FUNCTION_BLOCK FB_MatAndToolHandling EXTENDS FB_CompositionBase
VAR
	
	// Sequencer
	fbSeq						: FB_Sequence;
	
	stPosition					: ST_Coordinate;
	nToolDockingNr				: INT;
	
	fVelocityX					: LREAL;	
	fVelocityY					: LREAL;
	fAccelerationX				: LREAL;	
	fAccelerationY				: LREAL;
	
	bJogReverseDirectionX		: BOOL;
	bJogReverseDirectionY		: BOOL;
	bJogX						: BOOL;
	bJogY						: BOOL;
		
	bMoveX						: BOOL;
	bMoveY						: BOOL;
	
	// Watch Variables	
	refObstacle					: REFERENCE TO BOOL;
	bInPosition					: BOOL;
	
	// Tool/Mat Data
	nCurTooldockingNr			: INT;
	afDistanceTooldocking		: ARRAY[1..2] OF REAL;	
	astOffsetDie				: ARRAY[1..2] OF ST_Coordinate;
	

	nVelocityMultiplier			: INT;
	nAccelerationMultiplier		: INT;	
	stOffsetMat					: ST_Coordinate;
	
	
	// Settings
	
	fMaxVelocityX				: LREAL;
	fMinVelocityX				: LREAL;
	fMaxAccelerationX			: LREAL;
	fMinAccelerationX			: LREAL;
	
	fMaxVelocityY				: LREAL;
	fMinVelocityY				: LREAL;
	fMaxAccelerationY			: LREAL;
	fMinAccelerationY			: LREAL;
	
	fDefaultVelocity			: LREAL;
	fDefaultAcceleration		: LREAL;	
	
	fToleranceWindow			: LREAL := 0.5;
	stMaintPosition				: ST_Coordinate;
	
	// Axis
	bEnable						: BOOL := TRUE;
	refEnable					: REFERENCE TO BOOL;
	fbAxisX						: FB_AxisDriver;
	fbAxisY						: FB_AxisDriver;
	
	// Cylinder
	fbToolSelector				: FB_CylinderDriver;
	
END_VAR

METHOD _ChangeTool : BOOL
VAR_INPUT
END_VAR
fbSeq.Name := 'ChangeTool';

CASE fbSeq.Step OF
	

0	 :	fbSeq.StepDefinition('switch Valves for selected Tooldocking', T#0S);
		
		CASE nToolDockingNr OF
			1: fbToolSelector.ToWP();		
			2: fbToolSelector.ToHP();
		END_CASE

		fbSeq.NextStep(10);
	
	
10	 :	fbSeq.StepDefinition('Tooldock changing', T#0S);

		IF fbToolSelector.ActualPosition = fbToolSelector.RequestPosition THEN
			nCurTooldockingNr := nToolDockingNr;
			fbSeq.Finish();
		END_IF
	

END_CASE
END_METHOD

METHOD _Halt : BOOL
VAR_INPUT
END_VAR
fbSeq.Name := 'Halt';

CASE fbSeq.Step OF
	

0	 :	fbSeq.StepDefinition('Punchaxis Halt', T#0S);
		fbAxisX.Halt();
		fbAxisY.Halt();				
		fbSeq.NextStep(10);
	
	
10	 :	fbSeq.StepDefinition('', T#0S);
		IF fbAxisX.NotMoving AND fbAxisY.NotMoving THEN
			fbSeq.Finish();
		END_IF
	
END_CASE
END_METHOD

METHOD _Homeing : BOOL
VAR_INPUT
END_VAR
fbSeq.Name := 'Homeing';

CASE fbSeq.Step OF
	

0	 :	fbSeq.StepDefinition('', T#0S);

		fbSeq.NextStep(10);
	
	
10	 :	fbSeq.StepDefinition('', T#0S);

		fbSeq.NextStep(20);	

		
20	 :	fbSeq.StepDefinition('', T#0S);

		fbSeq.NextStep(30);	

		
30	 :	fbSeq.StepDefinition('', T#0S);

		fbSeq.NextStep(40);

		
40	 :	fbSeq.StepDefinition('', T#0S);

		fbSeq.NextStep(50);

		
50	 :	fbSeq.StepDefinition('', T#0S);

		fbSeq.Finish();

END_CASE
END_METHOD

METHOD _Jog : BOOL
VAR
	
END_VAR
fbSeq.Name := 'Jog';

CASE fbSeq.Step OF
	

0	 :	fbSeq.StepDefinition('Halt Axis', T#0S);
		fbAxisX.Halt();
		fbAxisY.Halt();	
		fbSeq.NextStep(10);
	
10	 :	fbSeq.StepDefinition('Jog Axis', T#0S);
	
		IF bJogX OR bJogY THEN
			fbAxisX.JogAcc(bJogX AND NOT bJogReverseDirectionX , bJogX AND bJogReverseDirectionX);
			fbAxisY.JogAcc(bJogY AND NOT bJogReverseDirectionY , bJogY AND bJogReverseDirectionY);
		ELSE
			fbSeq.NextStep(20);
		END_IF		
		
20	 :	fbSeq.StepDefinition('Jog Finish', T#0S);
		fbAxisX.Halt();
		fbAxisY.Halt();	
		fbSeq.Finish();

END_CASE
END_METHOD

METHOD _MoveAbs : BOOL
VAR
	stMovAbsParameter			: ST_AxisMoveAbsParameter;
END_VAR
fbSeq.Name := 'MoveAbs';

CASE fbSeq.Step OF
	

0	 :	fbSeq.StepDefinition('Move Axis to Position', T#0S);
		
		IF bMoveX THEN
			stMovAbsParameter.fAcceleration := fAccelerationX;
			stMovAbsParameter.fDeceleration := fAccelerationX;
			stMovAbsParameter.fVelocity := fVelocityX;
			stMovAbsParameter.fPosition := stPosition.fX;
			fbAxisX.MoveAbsEx(stMovAbsParameter);
		END_IF
			
		IF bMoveY THEN
			stMovAbsParameter.fAcceleration := fAccelerationY;
			stMovAbsParameter.fDeceleration := fAccelerationY;
			stMovAbsParameter.fVelocity := fVelocityY;
			stMovAbsParameter.fPosition := stPosition.fY;
			fbAxisY.MoveAbsEx(stMovAbsParameter);
		END_IF
		
		fbSeq.NextStep(20);	
		
20	 :	fbSeq.StepDefinition('Axis moving', T#0S);
		IF (fbAxisX.TargetReached(fToleranceWindow) OR NOT bMoveX) AND (fbAxisY.TargetReached(fToleranceWindow) OR NOT bMoveY) THEN
			fbSeq.Finish();
		END_IF

END_CASE
END_METHOD

/// Actual amplifier temp. [°C]
PROPERTY AmplifierTemp : LREAL
GET
/// Actual amplifier temp. [°C]
AmplifierTemp := MAX(fbAxisX.AmplifierTemp, fbAxisY.AmplifierTemp);
END_GET
END_PROPERTY

METHOD ChangeTool : E_OperationResult
VAR_INPUT
	ToolDockingNr				: INT;
END_VAR
// init result pessimistic
ChangeTool := E_OperationResult.eOperationResult_NOk;

bInPosition := FALSE;


stPosition := stMaintPosition;
fVelocityX := fVelocityY := fDefaultVelocity;	
fAccelerationX := fAccelerationY := fDefaultAcceleration;
nToolDockingNr := ToolDockingNr;
bMoveX := TRUE;
bMoveY := TRUE;

fbSeq.Start(E_MatAndToolHandlingCmd.cmdChangeTool);

ChangeTool := E_OperationResult.eOperationResult_Ok;
END_METHOD

PROPERTY CurTool : INT
GET
CurTool := nCurTooldockingNr;
END_GET
END_PROPERTY

METHOD FB_init : BOOL
VAR_INPUT
	bInitRetains : BOOL; // if TRUE, the retain variables are initialized (warm start / cold start)
	bInCopyCode : BOOL;  // if TRUE, the instance afterwards gets moved into the copy code (online change)
END_VAR
eTyp := E_ComponentType.eComponentType_MatAndToolHandling;
END_METHOD

METHOD GetMovementTime : LREAL
VAR_INPUT
	DistanceX		: LREAL;
	DistanceY		: LREAL;
	VelocityX		: LREAL;
	AccelerationX	: LREAL;
	VelocityY		: LREAL;
	AccelerationY	: LREAL;
END_VAR
VAR
	tmpTimeX		: LREAL;
	tmpTimeY		: LREAL;
	
	tmpTimeB		: LREAL;
	tmpTimeBB		: LREAL;
END_VAR
// X
tmpTimeB  := VelocityX/AccelerationX;
tmpTimeBB := 2*SQRT(DistanceX/AccelerationX);

IF tmpTimeBB/2 > tmpTimeB THEN
	tmpTimeX := DistanceX/VelocityX + VelocityX/AccelerationX;
ELSE
	tmpTimeX := tmpTimeBB;
END_IF


// Y
tmpTimeB  := VelocityY/AccelerationY;
tmpTimeBB := 2*SQRT(DistanceY/AccelerationY);

IF tmpTimeBB/2 > tmpTimeB THEN
	tmpTimeY := DistanceY/fVelocityY + VelocityY/AccelerationY;
ELSE
	tmpTimeY := tmpTimeBB;
END_IF


GetMovementTime := MAX(tmpTimeX, tmpTimeY)*1.2;	// 20% sicherheit
END_METHOD

METHOD Halt : E_OperationResult
VAR_INPUT
END_VAR
// init result pessimistic
Halt := E_OperationResult.eOperationResult_NOk;

bInPosition := FALSE;


fVelocityX := fVelocityY := fDefaultVelocity;	
fAccelerationX := fAccelerationY := fDefaultAcceleration;
bMoveX := FALSE;
bMoveY := FALSE;

fbSeq.Start(E_MatAndToolHandlingCmd.cmdHalt);

Halt := E_OperationResult.eOperationResult_Ok;
END_METHOD

PROPERTY Homed : BOOL
GET
Homed := fbaxisX.Homed AND fbaxisY.Homed;
END_GET
END_PROPERTY

METHOD Homing : E_OperationResult
VAR_INPUT
END_VAR
// init result pessimistic
Homing := E_OperationResult.eOperationResult_NOk;

bInPosition := FALSE;


stPosition := stMaintPosition;
fVelocityX := fVelocityY := fDefaultVelocity;	
fAccelerationX := fAccelerationY := fDefaultAcceleration;
bMoveX := TRUE;
bMoveY := TRUE;

fbSeq.Start(E_MatAndToolHandlingCmd.cmdHomeing);

Homing := E_OperationResult.eOperationResult_Ok;
END_METHOD

METHOD JogX : E_OperationResult
VAR_INPUT
	ReverseDirection					: BOOL;
END_VAR
// init result pessimistic
JogX := E_OperationResult.eOperationResult_NOk;
bInPosition := FALSE;

IF fbSeq.SequenceId <> E_MatAndToolHandlingCmd.cmdJog THEN
	fbSeq.Start(E_MatAndToolHandlingCmd.cmdJog);
//	RETURN;
END_IF


bJogReverseDirectionX := ReverseDirection;
bJogX := TRUE;	

JogX := E_OperationResult.eOperationResult_Ok;
END_METHOD

METHOD JogXStop : E_OperationResult
VAR_INPUT
END_VAR
// init result pessimistic
JogXStop := E_OperationResult.eOperationResult_NOk;

bJogX := FALSE;	

JogXStop := E_OperationResult.eOperationResult_Ok;
END_METHOD

METHOD JogY : E_OperationResult
VAR_INPUT
	ReverseDirection					: BOOL;
END_VAR
// init result pessimistic
JogY := E_OperationResult.eOperationResult_NOk;
bInPosition := FALSE;

IF fbSeq.SequenceId <> E_MatAndToolHandlingCmd.cmdJog THEN
	fbSeq.Start(E_MatAndToolHandlingCmd.cmdJog);
//	RETURN;
END_IF


bJogReverseDirectionY := ReverseDirection;
bJogY := TRUE;	

JogY := E_OperationResult.eOperationResult_Ok;
END_METHOD

METHOD JogYStop : E_OperationResult
VAR_INPUT
END_VAR
// init result pessimistic
JogYStop := E_OperationResult.eOperationResult_NOk;

bJogY := FALSE;	

JogYStop := E_OperationResult.eOperationResult_Ok;
END_METHOD

METHOD MaintPos : E_OperationResult
VAR_INPUT
	bXOnly				: BOOL;
	bYOnly				: BOOL;
END_VAR
IF bXOnly THEN
	MaintPos := MoveAbsX(stMaintPosition.fX,fDefaultVelocity, fDefaultAcceleration);	
ELSIF bYOnly THEN
	MaintPos := MoveAbsY(stMaintPosition.fY,fDefaultVelocity, fDefaultAcceleration);
ELSE
	MaintPos := MoveAbs(stMaintPosition,fDefaultVelocity, fDefaultAcceleration,fDefaultVelocity, fDefaultAcceleration);
END_IF


// override the calculated Position, Maintpos is independent of Tool
stPosition := stMaintPosition;
END_METHOD

/// Actual motor temp. [°C]
PROPERTY MotorTemp : LREAL
GET
/// Actual motor temp. [°C]
MotorTemp := MAX(fbAxisX.MotorTemp,fbAxisY.MotorTemp);
END_GET
END_PROPERTY

METHOD MoveAbs : E_OperationResult
VAR_INPUT
	Positon					: ST_Coordinate;
	VelocityX				: LREAL;
	AccelerationX			: LREAL;
	VelocityY				: LREAL;
	AccelerationY			: LREAL;
END_VAR
// init result pessimistic
MoveAbs := E_OperationResult.eOperationResult_NOk;

bInPosition := FALSE;

stPosition.fX := Positon.fX + stOffsetMat.fX ;//+ astOffsetDie[nCurTooldockingNr].fX
stPosition.fY := Positon.fY - afDistanceTooldocking[nCurTooldockingNr] + stOffsetMat.fY; //+ astOffsetDie[nCurTooldockingNr].fY 

// TODO: Check Coordinates if they are in/outside the traversing range

//IF ABS(fbAxisX.ActPos - stPosition.fX) < fToleranceWindow THEN
//	fVelocityY := MAX(MIN(fMaxVelocityY, VelocityY),fMinVelocityY);	
//	fAccelerationY := MAX(MIN(fMaxAccelerationY, AccelerationY),fMinAccelerationY);
//	bMoveX := FALSE;
//	bMoveY := TRUE;	
//ELSIF ABS(fbAxisY.ActPos - stPosition.fY) < fToleranceWindow THEN
//	fVelocityX := MAX(MIN(fMaxVelocityX, VelocityX),fMinVelocityX);	
//	fAccelerationX := MAX(MIN(fMaxAccelerationX, AccelerationX),fMinAccelerationX);
//	bMoveX := TRUE;
//	bMoveY := FALSE;
//ELSE	
	fVelocityY := MAX(MIN(fMaxVelocityY, VelocityY),fMinVelocityY);	
	fAccelerationY := MAX(MIN(fMaxAccelerationY, AccelerationY),fMinAccelerationY);
	fVelocityX := MAX(MIN(fMaxVelocityX, VelocityX),fMinVelocityX);	
	fAccelerationX := MAX(MIN(fMaxAccelerationX, AccelerationX),fMinAccelerationX);
	bMoveX := TRUE;
	bMoveY := TRUE;
	
//END_IF

fbSeq.Start(E_MatAndToolHandlingCmd.cmdMoveAbs);

MoveAbs := E_OperationResult.eOperationResult_Ok;
END_METHOD

METHOD MoveAbsX : E_OperationResult
VAR_INPUT
	Positon					: REAL;
	Velocity				: LREAL;
	Acceleration			: LREAL;
END_VAR
// init result pessimistic
MoveAbsX := E_OperationResult.eOperationResult_NOk;

bInPosition := FALSE;

stPosition := THIS^.Position;
stPosition.fX := Positon;
fVelocityX := MAX(MIN(fMaxVelocityX, Velocity),fMinVelocityX);	
fAccelerationX := MAX(MIN(fMaxAccelerationX, Acceleration),fMinAccelerationX);
bMoveX := TRUE;
bMoveY := FALSE;

fbSeq.Start(E_MatAndToolHandlingCmd.cmdMoveAbs);

MoveAbsX := E_OperationResult.eOperationResult_Ok;
END_METHOD

METHOD MoveAbsY : E_OperationResult
VAR_INPUT
	Positon					: REAL;
	Velocity				: LREAL;
	Acceleration			: LREAL;
END_VAR
// init result pessimistic
MoveAbsY := E_OperationResult.eOperationResult_NOk;

bInPosition := FALSE;

stPosition := THIS^.Position;
stPosition.fY := Positon;
fVelocityY := MAX(MIN(fMaxVelocityY, Velocity),fMinVelocityY);	
fAccelerationY := MAX(MIN(fMaxAccelerationY, Acceleration),fMinAccelerationY);
bMoveX := FALSE;
bMoveY := TRUE;

fbSeq.Start(E_MatAndToolHandlingCmd.cmdMoveAbs);

MoveAbsY := E_OperationResult.eOperationResult_Ok;
END_METHOD

METHOD MoveRelX : E_OperationResult
VAR_INPUT
	Distance				: LREAL;
	Velocity				: LREAL;
	Acceleration			: LREAL;
END_VAR

VAR
	tmpPos					: ST_Coordinate;
END_VAR
// init result pessimistic
MoveRelX := E_OperationResult.eOperationResult_NOk;

bInPosition := FALSE;

tmpPos := Position;
tmpPos.fX := MAX(fbAxisX.LimitNeg, MIN(fbAxisX.LimitPos, tmpPos.fX + Distance));

stPosition := tmpPos;
fVelocityX := MAX(MIN(fMaxVelocityX, Velocity),fMinVelocityX);	
fAccelerationX := MAX(MIN(fMaxAccelerationX, Acceleration),fMinAccelerationX);
bMoveX := TRUE;
bMoveY := FALSE;

fbSeq.Start(E_MatAndToolHandlingCmd.cmdMoveAbs);

MoveRelX := E_OperationResult.eOperationResult_Ok;
END_METHOD

METHOD MoveRelY : E_OperationResult
VAR_INPUT
	Distance				: LREAL;
	Velocity				: LREAL;
	Acceleration			: LREAL;
END_VAR

VAR
	tmpPos					: ST_Coordinate;
END_VAR
// init result pessimistic
MoveRelY := E_OperationResult.eOperationResult_NOk;

bInPosition := FALSE;

tmpPos := Position;
tmpPos.fY := MAX(fbAxisY.LimitNeg, MIN(fbAxisY.LimitPos, tmpPos.fY + Distance));;

stPosition := tmpPos;
fVelocityY := MAX(MIN(fMaxVelocityY, Velocity),fMinVelocityY);	
fAccelerationY := MAX(MIN(fMaxAccelerationY, Acceleration),fMinAccelerationY);
bMoveX := FALSE;
bMoveY := TRUE;

fbSeq.Start(E_MatAndToolHandlingCmd.cmdMoveAbs);

MoveRelY := E_OperationResult.eOperationResult_Ok;
END_METHOD

PROPERTY Moving : BOOL
GET
Moving := fbAxisX.Moving OR fbAxisY.Moving;
END_GET
END_PROPERTY

PROPERTY NotMoving : BOOL
GET
NotMoving := NOT Moving;
END_GET
END_PROPERTY

PROPERTY Override : LREAL
GET
Override := MAX(fbAxisX.Override, fbAxisY.Override);
END_GET
SET
fbAxisX.Override := Override;
fbAxisY.Override := Override;
END_SET
END_PROPERTY

PROPERTY Position : ST_Coordinate
GET
Position.fX := fbAxisX.Position;
Position.fY := fbAxisY.Position;
END_GET
END_PROPERTY

PROPERTY Ready : BOOL
GET
Ready := fbAxisX.MotionState <> MC_AXISSTATE_DISABLED AND fbAxisY.MotionState <> MC_AXISSTATE_DISABLED;
END_GET
END_PROPERTY

/// Reset component logic
{attribute 'object_name' := 'Reset'}
METHOD Reset
// base logic run
SUPER^.Reset();

fbAxisY.Reset();
fbAxisX.Reset();

fbSeq.Init();
END_METHOD

/// Run component logic
{attribute 'object_name' := 'Run'}
METHOD Run : E_ComponentState
// run Base Logic
Run := SUPER^.Run();

IF __ISVALIDREF(refEnable) THEN
	bEnable := refEnable;
END_IF

// run Axis Driver
fbAxisX.Run();
fbAxisX.Enable := bEnable;
fbAxisX.EnablePos := bEnable;
fbAxisX.EnableNeg := bEnable;

fbAxisY.Run();
fbAxisY.Enable := bEnable;
fbAxisY.EnablePos := bEnable;
fbAxisY.EnableNeg := bEnable;

// run Cylinder Driver
fbToolSelector.Run();
fbToolSelector.SafetyOk := bEnable;
fbToolSelector.bEnableHp := bEnable;
fbToolSelector.bEnableWp := bEnable;


// run Sequences
fbSeq.Enable := TRUE;
fbSeq.Base(FALSE, FALSE);
CASE fbSeq.SequenceId OF	
	E_MatAndToolHandlingCmd.cmdMoveAbs:			_MoveAbs();
	E_MatAndToolHandlingCmd.cmdHalt:			_Halt();	
	E_MatAndToolHandlingCmd.cmdChangeTool:		_ChangeTool();	
	E_MatAndToolHandlingCmd.cmdJog:				_Jog();
	E_MatAndToolHandlingCmd.cmdHomeing:			_Homeing();
END_CASE
END_METHOD

METHOD Setup : BOOL
VAR_INPUT
	eAxis_X					: E_Axis;
	eAxis_Y					: E_Axis;
	eToolSelector		    : E_Cylinder;
END_VAR
fbAxisX.Name := 'X-Axis';
fbAxisX.SetAxisReference(COMP.astAxisRef[eAxis_X], COMP.astAxisIO[eAxis_X].stIn, COMP.astAxisIO[eAxis_X].stOut);
fbAxisX.AxisType := E_AxisType.AX5xxx;
fbAxisX.DefaultParameter.stMovAbsPrm.fVelocity := 30;
fbAxisX.Active := TRUE;
fbAxisX.Override := 100;
fbAxisX.DefaultParameter.stJogAccPrm.fFastSpeed := 240;
fbAxisX.DefaultParameter.stJogAccPrm.fSlowSpeed := 10;
fbAxisX.DefaultParameter.stJogAccPrm.tAccTime := T#5S;
fbAxisX.SetSecondPosFeedback(3640, 3.9630466037326388888888888888889E-5);
fbAxisX.EnableLimitSensor:= FALSE;	
fbAxisX.LimitNeg := 10;
fbAxisX.LimitPos := 4070;

fbAxisY.Name := 'Y-Axis';
fbAxisY.SetAxisReference(COMP.astAxisRef[eAxis_Y], COMP.astAxisIO[eAxis_Y].stIn, COMP.astAxisIO[eAxis_Y].stOut);
fbAxisY.AxisType := E_AxisType.AX5xxx;
fbAxisY.DefaultParameter.stMovAbsPrm.fVelocity := 30;
fbAxisY.Active := TRUE;
fbAxisX.Override := 100;
fbAxisY.DefaultParameter.stJogAccPrm.fFastSpeed := 240;
fbAxisY.DefaultParameter.stJogAccPrm.fSlowSpeed := 10;
fbAxisY.DefaultParameter.stJogAccPrm.tAccTime := T#5S;
fbAxisY.EnableLimitSensor:= FALSE;	
fbAxisY.LimitNeg := 5;
fbAxisY.LimitPos := 790;

fbToolSelector.Name := 'Zylinder';
fbToolSelector.SetIoReference(aStCylinderIO[eToolSelector].stIn, aStCylinderIO[eToolSelector].stOut);
fbToolSelector.EnableHpSensor := TRUE;
fbToolSelector.EnableWpSensor := TRUE;
//fbToolSelector.SetImpulseTime := 
//fbToolSelector.PositionValidationTime :=


fMaxVelocityX			:= 4700;
fMinVelocityX			:= 10;
fMaxAccelerationX		:= 10000;
fMinAccelerationX		:= 0;
fMaxVelocityY			:= 3200;
fMinVelocityY			:= 10;
fMaxAccelerationY		:= 10000;
fMinAccelerationY		:= 0;
fDefaultVelocity		:= 100;
fDefaultAcceleration	:= 0;
fToleranceWindow		:= 0.5;
END_METHOD

METHOD SetupEnable : BOOL

VAR_IN_OUT
	bEnable					: BOOL;
END_VAR
refEnable REF= bEnable;
END_METHOD

METHOD SetupMaintPos : BOOL
VAR_INPUT
	MaintPosition		: ST_Coordinate;
END_VAR
stMaintPosition	:=  MaintPosition;
END_METHOD

METHOD SetupMat : BOOL
VAR_INPUT
	Offset			: ST_Coordinate;
END_VAR
stOffsetMat:= Offset;
END_METHOD

METHOD SetupObstacle : BOOL
VAR_IN_OUT
	Obstacle			: BOOL;
END_VAR
refObstacle REF= Obstacle;
END_METHOD

METHOD SetupToolDistance : BOOL
VAR_INPUT
	fDistanceToolDock1		: REAL;
	fDistanceToolDock2		: REAL;
END_VAR
afDistanceTooldocking[1]	:=  fDistanceToolDock1;
afDistanceTooldocking[2]	:=  fDistanceToolDock2;
END_METHOD

METHOD SetupToolholder : BOOL
VAR_INPUT
	DockingNr		: INT;
	fDieOffsetX		: REAL;
	fDieOffsetY		: REAL;
END_VAR
astOffsetDie[DockingNr].fX := fDieOffsetX;
astOffsetDie[DockingNr].fY := fDieOffsetY;
END_METHOD

{attribute 'monitoring' := 'variable'}
PROPERTY TargetReached : BOOL
GET
TargetReached := fbAxisX.TargetReached(fToleranceWindow) AND fbAxisY.TargetReached(fToleranceWindow);
END_GET
END_PROPERTY

PROPERTY ToolChanged : BOOL
GET
ToolChanged := nCurTooldockingNr = nToolDockingNr;
END_GET
END_PROPERTY

/// The torque limit for both directions. [Nm]
PROPERTY TorqueLimitX : LREAL
GET
/// The torque limit for both directions. [1/10%]
TorqueLimitX := fbAxisX.TorqueLimit;
END_GET
SET
fbAxisX.TorqueLimit := TorqueLimitX;
END_SET
END_PROPERTY

/// The torque limit for both directions. [Nm]
PROPERTY TorqueLimitY : LREAL
GET
/// The torque limit for both directions. [1/10%]
TorqueLimitY := fbAxisY.TorqueLimit;
END_GET
SET
fbAxisY.TorqueLimit := TorqueLimitY;
END_SET
END_PROPERTY

END_FUNCTION_BLOCK

(* stored: Version 1.1.0.1, ProductVersion 3.1.4022.12
   POU FB_MatAndToolHandling: Id {a6bb103e-ddbd-41c7-9d04-5c7fca296ec9}, SpecialFunc None
   Folder Commands: Id {377f9c91-d0c7-42d8-951e-ff1d956d437a}
   Folder Properties: Id {658f387c-1b3c-422b-8b15-9aa5381860ec}
   Folder Sequences: Id {cd7652ee-8198-4eed-861a-a7ed543e0f62}
   Folder Setup: Id {ae65bc78-5fd6-47e0-96e6-e84065484636}
   Folder Utilities: Id {cd021480-2e63-4703-8886-72b16ef7094f}
   Method _ChangeTool: Id {f0ab3374-31e9-4529-8c12-c3506d2f5919}
   Method _Halt: Id {6e59e6b5-773f-4790-89cb-2010bd373a91}
   Method _Homeing: Id {a56b25bb-fe72-44dc-80b5-637f2fcb4907}
   Method _Jog: Id {1d2ff23e-33f0-4a92-b3b2-26e22dd33108}
   Method _MoveAbs: Id {4bfcd30e-7191-4dcc-a300-81025d11d7f1}
   Property AmplifierTemp: Id {a44d240b-0646-4f6d-bf88-e30572090b8f}
   Get Get: Id {9adf4361-d80a-473b-b4b7-eb470cf7138d}
   Method ChangeTool: Id {c588bd96-44d3-43fa-8ba5-9bf373d5e2bc}
   Property CurTool: Id {b0b358e0-e403-4312-a7e4-0b60a25569a2}
   Get Get: Id {6479b220-a466-4b93-8696-18abdad3aca2}
   Method FB_init: Id {e1ed02d3-3c8c-4424-815c-632247250740}
   Method GetMovementTime: Id {c1482001-afc0-4aba-b421-809c696fd43d}
   Method Halt: Id {92f2c6c9-156d-4bca-9b55-fe2aca91bd9b}
   Property Homed: Id {c9d61529-2cd7-4b34-941c-55aca463530f}
   Get Get: Id {9737d753-e7f1-459b-b948-78edc9855295}
   Method Homing: Id {22980133-2b13-41f4-b814-e48099b58c9b}
   Method JogX: Id {b043ecd2-382c-4f85-8b01-ac75c7b03c3e}
   Method JogXStop: Id {6fe34396-2950-4a93-b24f-960f3bfac0f9}
   Method JogY: Id {c5453b2b-6337-49d6-a443-484ca70fbfe0}
   Method JogYStop: Id {f1d239eb-ac84-41a8-8f1e-6767a2a6c9ab}
   Method MaintPos: Id {7a877f5e-256c-417b-a796-2359094340b8}
   Property MotorTemp: Id {c05b9444-a31f-43a7-b77e-03039c6c3f0f}
   Get Get: Id {efeb379c-d6b4-4b78-ba41-237a43755ad5}
   Method MoveAbs: Id {a109d053-4806-4f10-b44b-e30d01f0a7b3}
   Method MoveAbsX: Id {c8d45f91-e2c3-4159-a4f7-a6628b762024}
   Method MoveAbsY: Id {76efc827-2a40-45c4-92dc-25f66feab386}
   Method MoveRelX: Id {ecaed027-789b-4c6c-b40f-ac25d95aeeb5}
   Method MoveRelY: Id {732ef1f1-c1c0-4ace-98ba-e2ffc7fb86ac}
   Property Moving: Id {0dce4285-d95e-436e-bd27-e2f7edcbe838}
   Get Get: Id {98b10ba6-9d5b-4af6-bb57-d493e47fccec}
   Property NotMoving: Id {1e706dca-279f-4a63-a593-040719d331d7}
   Get Get: Id {b56bf59e-892e-4223-a22a-2ec8f7c89428}
   Property Override: Id {75fcc446-a1e6-400d-9052-f66c52e0328b}
   Get Get: Id {b80ea9cd-c316-4a72-96ea-0f6958434ef7}
   Set Set: Id {95c2e620-6254-4c8c-876f-3e0b9afadc37}
   Property Position: Id {6e649e63-b55e-47e6-93ad-e3a6abdb271d}
   Get Get: Id {91c845b6-a1d7-4020-ba3a-e0dc9c3c4c4b}
   Property Ready: Id {927ed93f-f291-463e-8286-93bfa26d321a}
   Get Get: Id {50cac311-dfaa-42a0-b252-f4491661bb2f}
   Method Reset: Id {6d37851e-e615-43b8-b8ff-783e7579ef72}
   Method Run: Id {c9018ee7-bbca-46a8-be5f-0c5efcbdc5bc}
   Method Setup: Id {f607b703-6908-4869-8c11-943de5cbe8eb}
   Method SetupEnable: Id {d80a8f5a-3eca-4da0-a90b-4cfeb95f54da}
   Method SetupMaintPos: Id {484665e7-c6bc-44df-87b6-cf024c838db6}
   Method SetupMat: Id {04eaa570-e65e-4393-8b32-1de476ed9a3b}
   Method SetupObstacle: Id {f48a94ac-b2e3-40d6-b8c7-dbbba451e3d3}
   Method SetupToolDistance: Id {cdc79598-c0f1-4f99-bf24-e142dee8c62c}
   Method SetupToolholder: Id {a886c911-57a8-430d-9d73-4c723d008686}
   Property TargetReached: Id {c5d24c72-4827-4293-b4ba-08994b17ca63}
   Get Get: Id {7e5d009f-904a-4223-85e4-a6deb5534aa8}
   Property ToolChanged: Id {e7e4f597-ca3b-4956-9ee0-8f39af4943af}
   Get Get: Id {79c818fe-3899-49d4-bc93-802802dd64ea}
   Property TorqueLimitX: Id {9334d840-cb87-4b0a-85ec-7c5362e76f58}
   Get Get: Id {3f5d3134-733e-45d2-896e-ac35c05d70bf}
   Set Set: Id {d679d6d9-7094-4bba-aa53-1856d247e4a2}
   Property TorqueLimitY: Id {1a03d889-f029-475b-80d4-16f537f3e5c7}
   Get Get: Id {76ef9422-533b-409c-8866-aad1e2c4b334}
   Set Set: Id {4d958039-0647-46cc-87e4-bc4ba3ba1de8} *)
